ABB RobotStudio station: burguerBotVentosaYSensores.rspag

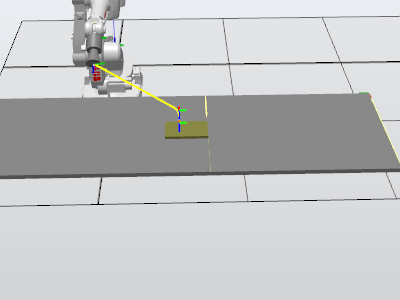
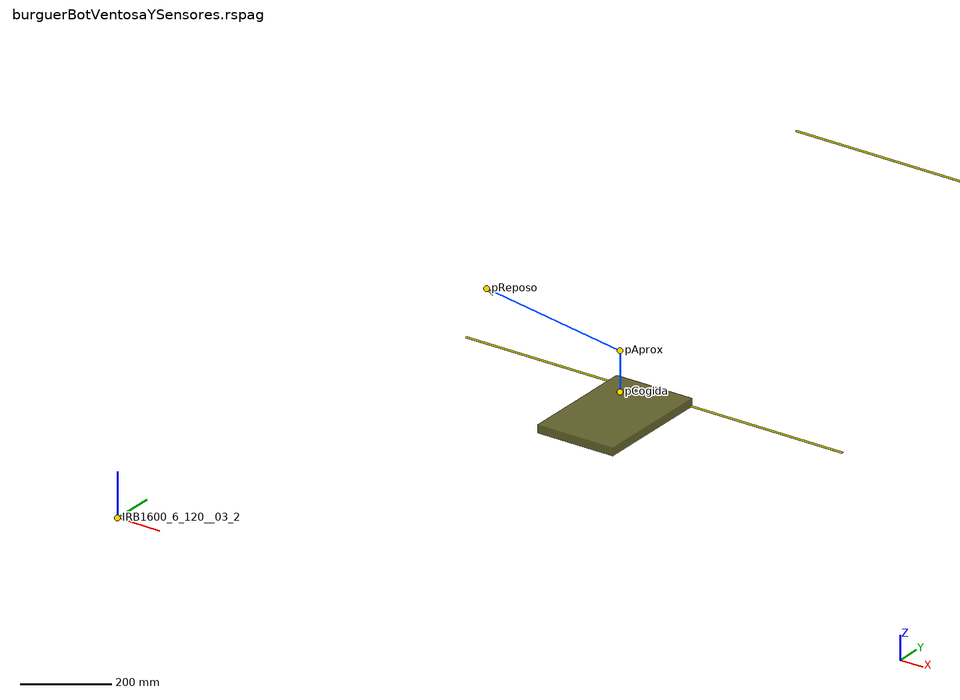
[picture v1: parts stored in the station drawn from their meshes, with robot base, taught points and paths (robot models come from the ABB library and are not in the file)]
--- station ---
Station Station (saved by RobotStudio 24.1.10713.1)
Controller Controlador4, task T_ROB1: task frame (RAPID world) sits at (600, 0, 0) mm in the station
Controller Controlador4
  mechanical unit ROB_1: IRB1600_6_120__03_2, 6 joints, base frame (0, 0, 0) mm
Layout (positions relative to the parent item):
  - Ventosa [mechanism, from Libraries\Ventosa.rslib] at (1406.29, 0, 929) mm, rotated rx 180 ry 60 rz 180 deg
  - CintaTransportadora [part, from Libraries\CintaTransportadora.rslib] at (0, 0, -500) mm
  - IRB1600_6_120__03_2 [mechanism, from %ABB.RobotStudio.Models.IRB1600%\IRB1600_6_120_G_03.rslib] at (600, 0, 0) mm; joint values [0, 0, 0, 0, 0.5236, 0] (rad or m)
  - SmartComponent_2 [smart component]
      signals: DO PiezaDetectada, DI ActivaVentosa, DO Vacuostato
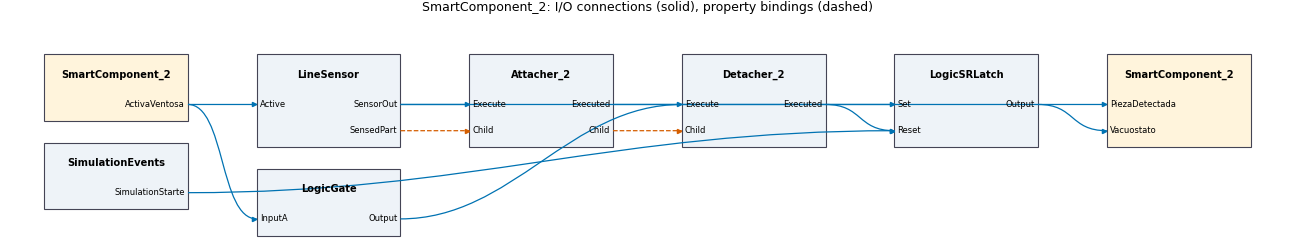
      connections:
        SmartComponent_2.ActivaVentosa -> LineSensor.Active
        SmartComponent_2.ActivaVentosa -> LogicGate.InputA
        LogicGate.Output -> Detacher_2.Execute
        LineSensor.SensorOut -> Attacher_2.Execute
        LineSensor.SensorOut -> SmartComponent_2.PiezaDetectada
        Attacher_2.Executed -> LogicSRLatch.Set
        Detacher_2.Executed -> LogicSRLatch.Reset
        SimulationEvents.SimulationStarted -> LogicSRLatch.Reset
        LogicSRLatch.Output -> SmartComponent_2.Vacuostato
        Attacher_2.Child => Detacher_2.Child
        LineSensor.SensedPart => Attacher_2.Child
    - LineSensor [smart component, from Components\LineSensor.rslib] at (1579.5, 0, 829) mm, rotated rx 180 ry 60 rz 180 deg
        properties: Start=[0 0 -0.002]; End=[0 0 0.02]; Length=0.022; Radius=0.002; Tag=(none); SensedPart=(none); SensedPoint=[1.55 0.549999938964844 0.35]
      - _sensorPart_ [part], size 4 x 4 x 22 mm
    - SimulationEvents [smart component, from Components\SimulationEvents.rslib]
    - LogicSRLatch [smart component, from Components\LogicSRLatch.rslib]
    - Attacher_2 [smart component, from Components\Attacher.rslib]
        properties: Parent=Ventosa; Flange=0; Child=(none); Mount=false; Offset=[0 0 0]; Orientation=[0 0 0]
    - Detacher_2 [smart component, from Components\Detacher.rslib]
        properties: Child=(none); KeepPosition=true
    - LogicGate [smart component, from Components\LogicGate.rslib]
        properties: Operator=NOT; Delay=0
  - CI_SensoresCinta [smart component] at (0, 0, -500) mm
      signals: DI ActivaSensores, DO BandejaEnPos, DO FinalCinta
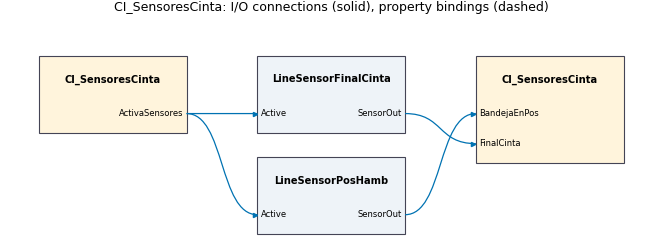
      connections:
        CI_SensoresCinta.ActivaSensores -> LineSensorFinalCinta.Active
        CI_SensoresCinta.ActivaSensores -> LineSensorPosHamb.Active
        LineSensorPosHamb.SensorOut -> CI_SensoresCinta.BandejaEnPos
        LineSensorFinalCinta.SensorOut -> CI_SensoresCinta.FinalCinta
    - LineSensorFinalCinta [smart component, from Components\LineSensor.rslib]
        properties: Start=[2 2 0.75]; End=[1 2 0.75]; Length=1; Radius=0.002; Tag=(none); SensedPart=CintaTransportadora; SensedPoint=[1 2 0.25]
      - _sensorPart_ [part], size 1000 x 4 x 4 mm
    - LineSensorPosHamb [smart component, from Components\LineSensor.rslib]
        properties: Start=[2 0.75 0.75]; End=[1 0.75 0.75]; Length=1; Radius=0.002; Tag=(none); SensedPart=(none); SensedPoint=[0 0 0]
      - _sensorPart_ [part], size 1000 x 4 x 4 mm
  - Pieza_3 [part], size 1050 x 3000 x 100 mm
  - Pieza_7 [part], size 200 x 300 x 20 mm
Attachment: Ventosa is attached to IRB1600_6_120__03_2 / Link6
Attachment: LineSensor is attached to Ventosa / PiezaVentosa
Attachment: CI_SensoresCinta is attached to CintaTransportadora
Station logic (signal -> signal, property => property):
  SmartComponent_2.PiezaDetectada -> Controlador4.ED_PiezaDetectada
  Controlador4.SD_ActivaVentosa -> SmartComponent_2.ActivaVentosa
  SmartComponent_2.Vacuostato -> Controlador4.ED_PiezaCogida
Targets, tools, work objects and paths stored in the station and not in the controller backup, written as RAPID:
! task T_ROB1
MODULE Module1
  CONST robtarget Target_10:=[[579.496732003,2000,-579],[0,0.5,0,0.866025404],[0,0,0,0],[9E+09,9E+09,9E+09,9E+09,9E+09,9E+09]];
ENDMODULE


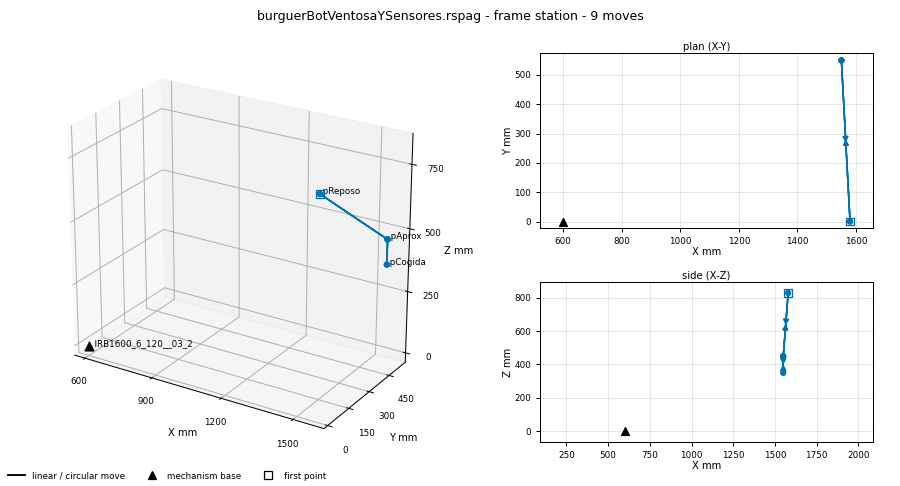
[picture p0: tool path of burguerBotVentosaYSensores.rspag in frame station, 9 of 9 moves have a stored position in this frame; points joined in program order, loops and branches not executed]
--- Backups/Controlador4/RAPID/TASK1/PROGMOD/CalibData.mod ---
MODULE CalibData
    PERS tooldata Ventosa:=[TRUE,[[0,0,200],[1,0,0,0]],[1,[0,0,125],[1,0,0,0],0.002,0.002,0.0013]];
    TASK PERS wobjdata Workobject_1:=[FALSE,TRUE,"",[[400,2000,250],[0,1,0,0]],[[0,0,0],[1,0,0,0]]];
ENDMODULE

--- Backups/Controlador4/RAPID/TASK1/PROGMOD/Module1.mod ---
MODULE Module1
        CONST robtarget pReposo:=[[979.496732003,0,829],[0.5,0,0.866025404,0],[0,0,-1,0],[9E+09,9E+09,9E+09,9E+09,9E+09,9E+09]];
    CONST robtarget pAprox:=[[550,1450,-200],[0,0,0,1],[0,0,0,0],[9E+09,9E+09,9E+09,9E+09,9E+09,9E+09]];
    CONST robtarget pCogida:=[[550,1450,-100],[0,0,0,1],[0,0,0,0],[9E+09,9E+09,9E+09,9E+09,9E+09,9E+09]];
!***********************************************************
    !
    ! M?dulo:  Module1
    !
    ! Descripción:
    !   <Introduzca la descripción aquí>
    !
    ! Autor: rafac
    !
    ! Versión: 1.0
    !
    !***********************************************************


    !***********************************************************
    !
    ! Procedimiento Main
    !
    !   Este es el punto de entrada de su programa
    !
    !***********************************************************
    PROC main()
        !Add your code here
        Path_20;
    ENDPROC
    PROC Path_20()
        MoveL pReposo,v1000,fine,Ventosa\WObj:=wobj0;
        MoveL pAprox,v1000,fine,Ventosa\WObj:=Workobject_1;
        MoveL pCogida,v1000,fine,Ventosa\WObj:=Workobject_1;
        SetDO SD_ActivaVentosa,1;
        WaitDi ED_PiezaCogida,1;
        MoveL pAprox,v1000,fine,Ventosa\WObj:=Workobject_1;
        MoveL pReposo,v1000,fine,Ventosa\WObj:=wobj0;
        MoveL pAprox,v1000,fine,Ventosa\WObj:=Workobject_1;
        MoveL pCogida,v1000,fine,Ventosa\WObj:=Workobject_1;
        SetDO SD_ActivaVentosa,0;
        WaitDI ED_PiezaCogida,0;
        MoveL pAprox,v1000,fine,Ventosa\WObj:=Workobject_1;
        MoveL pReposo,v1000,fine,Ventosa\WObj:=wobj0;

    ENDPROC
ENDMODULE

--- Backups/Controlador4/SYSPAR/EIO.cfg ---
EIO:CFG_1.0:6:1::
#
INDUSTRIAL_NETWORK:

      -Name "DeviceNet" -Label "DeviceNet Master/Slave Network" -Address "2"
#
DEVICENET_DEVICE:

      -Name "MiDeviceNet"
#
DEVICENET_INTERNAL_DEVICE:

      -Name "DN_Internal_Device" -VendorName "ABB Robotics"\
      -ProductName "DeviceNet Internal Slave Device"
#
EIO_SIGNAL:

      -Name "ED_PiezaDetectada" -SignalType "DI" -Device "MiDeviceNet"\
      -Label "ED_PiezaDetectada" -DeviceMap "0" -Access "All"

      -Name "ED_PiezaCogida" -SignalType "DI" -Device "MiDeviceNet"\
      -Label "ED_PiezaCogida" -DeviceMap "1" -Access "All"

      -Name "SD_ActivaVentosa" -SignalType "DO" -Device "MiDeviceNet"\
      -Label "SD_ActivaVentosa" -DeviceMap "0" -Access "All"
